FUNCTION_BLOCK controller
  (* Standard: 61499-2 *)
  (* Version 0.1, 2017-00-25, hpea485, UOA *)
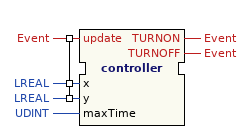
  EVENT_INPUT
    update WITH x, y;
  END_EVENT
  EVENT_OUTPUT
    TURNON;
    TURNOFF;
  END_EVENT
  VAR_INPUT
    x : LREAL;
    y : LREAL;
    maxTime : UDINT := 999;
  END_VAR
  VAR
    timer : UDINT := 0;
  END_VAR
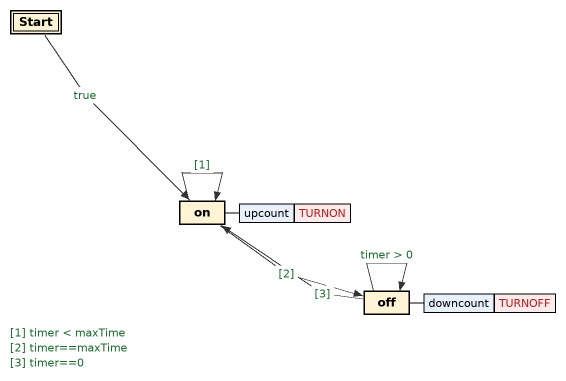
  EC_STATES
    Start;
    on : upcount -> TURNON;
    off : downcount -> TURNOFF;
  END_STATES
  EC_TRANSITIONS
    Start TO on := true;
    on TO off := timer==maxTime;
    on TO on := timer < maxTime;
    off TO on := timer==0;
    off TO off := timer > 0;
  END_TRANSITIONS
  ALGORITHM upcount IN C:
me->timer++;
if(me->timer > me->maxTime) {
	me->timer = me->maxTime;
}
  END_ALGORITHM
  ALGORITHM downcount IN C:
me->timer--;
if(me->timer < 0) {
	me->timer = 0;
}
  END_ALGORITHM
END_FUNCTION_BLOCK
